(* IEC 61131-3 sources: axftcmlib/src/Actuator, 6 files *)

(* ---- ActuatorStates.st ---- *)
NAMESPACE Simatic.Ax.axftcmlib
    TYPE
        ActuatorState : (Retracted, Activating, Activated, Retracting) := Retracted;
    END_TYPE
END_NAMESPACE

(* ---- IActuator.st ---- *)
USING Simatic.Ax.Commands;
NAMESPACE Simatic.Ax.axftcmlib
    INTERFACE IActuator
        METHOD Start : itfCommand END_METHOD
    END_INTERFACE
END_NAMESPACE

(* ---- itfActuator.st ---- *)
USING Simatic.Ax.Commands;

NAMESPACE Simatic.Ax.axftcmlib

    INTERFACE itfActuator
        METHOD GoToWorkPosition : itfCommand
        END_METHOD
    END_INTERFACE

    INTERFACE itfTwoWayActuator EXTENDS itfActuator
        METHOD GoToHomePosition : itfCommand
        END_METHOD
    END_INTERFACE

END_NAMESPACE

(* ---- ActuatorTimeBased.st ---- *)
USING Simatic.Ax.Commands;
USING System.Timer;
USING Simatic.Ax.Io.Output;

NAMESPACE Simatic.Ax.axftcmlib
    CLASS ActuatorTimeBased
        EXTENDS ExecuteControlModuleAbstract
        IMPLEMENTS itfActuator
        VAR PUBLIC
            Q_ToWorkPosition : IBinOutput;
            OnDuration : TIME;
        END_VAR
        VAR
            _tonOnDuration : OnDelay;
            _state : ActuatorState;
        END_VAR

        METHOD PROTECTED OVERRIDE _initmethod
            ;
        END_METHOD

        METHOD PROTECTED OVERRIDE _executeCustom
            IF (Q_ToWorkPosition = NULL) THEN
                THIS.SetError(WORD#16#8101);
                RETURN;
            ELSE
                THIS.SetError(FALSE);
            END_IF;
            _tonOnDuration(signal := Q_ToWorkPosition.IsOn(), Duration := OnDuration);
            CASE _state OF
                // Switch all outputs off, when actuator is idle in home position
                ActuatorState#InHomePosition:
                    Q_ToWorkPosition.SetOff();

                // Received the command GoToWorkPosition switch on ToWorkPosition
                ActuatorState#MoveToWorkPosition:
                    Q_ToWorkPosition.SetOn();
                    _state := ActuatorState#InWorkPosition;
                // After Timeout switch off "ToWorkPosition"
                ActuatorState#InWorkPosition:
                    IF (_tonOnDuration.output) THEN
                        _state := ActuatorState#MoveToHomePosition;
                        Q_ToWorkPosition.SetOff();
                    END_IF;
                // Send done
                ActuatorState#MoveToHomePosition:
                    Q_ToWorkPosition.SetOff();
                    _state := ActuatorState#InHomePosition;
                    THIS.SetDone();
            END_CASE;
        END_METHOD

        METHOD PUBLIC GoToWorkPosition : itfCommand
            THIS.InitState();
            _state := ActuatorState#MoveToWorkPosition;
            GoToWorkPosition := THIS;
        END_METHOD

        METHOD PUBLIC GetState : ActuatorState
            GetState := _state;
        END_METHOD

    END_CLASS

END_NAMESPACE

(* ---- TimeBasedActuator.st ---- *)
USING Simatic.Ax.Commands;
USING System.Timer;
USING Simatic.Ax.Io.Output;

NAMESPACE Simatic.Ax.axftcmlib

    CLASS TimeBasedActuator
        EXTENDS ExecuteControlModuleAbstract
        IMPLEMENTS itfActuator
        VAR PUBLIC
            Q_ToWorkPosition : ItfBinOutput;
            OnDuration : TIME;
        END_VAR
        VAR
            _tonOnDuration : OnDelay;
            _state : ActuatorState;
        END_VAR

        METHOD PROTECTED OVERRIDE _initmethod
            ;
        END_METHOD

        METHOD PROTECTED OVERRIDE _executeCustom
            IF (Q_ToWorkPosition = NULL) THEN
                THIS.SetError(WORD#16#8101);
                RETURN;
            END_IF;
            _tonOnDuration(signal := Q_ToWorkPosition.IsOn(), Duration := OnDuration);
            CASE _state OF
// Switch all outputs off, when actuator is idle in home position
                ActuatorState#InHomePosition:
                    Q_ToWorkPosition.SetOff();
// Received the command GoToWorkPosition switch on ToWorkPosition
                ActuatorState#MoveToWorkPosition:
                    Q_ToWorkPosition.SetOn();
                    _state := ActuatorState#InWorkPosition;
// After Timeout switch off "ToWorkPosition"
                ActuatorState#InWorkPosition:
                    IF (_tonOnDuration.output) THEN
                        _state := ActuatorState#MoveToHomePosition;
                        Q_ToWorkPosition.SetOff();
                    END_IF;
// Send done
                ActuatorState#MoveToHomePosition:
                    Q_ToWorkPosition.SetOff();
                    _state := ActuatorState#InHomePosition;
                    THIS.SetDone();
            END_CASE;
        END_METHOD

        METHOD PUBLIC GoToWorkPosition : itfCommand
            THIS.InitState();
            _state := ActuatorState#MoveToWorkPosition;
            GoToWorkPosition := THIS;
        END_METHOD

        METHOD PUBLIC GetState : ActuatorState
            GetState := _state;
        END_METHOD
    END_CLASS

END_NAMESPACE

(* ---- TwoWayActuator.st ---- *)
USING Simatic.Ax.IO.Input;
USING Simatic.Ax.Commands;
USING System.Timer;
USING Simatic.Ax.Io.Output;

NAMESPACE Simatic.Ax.axftcmlib

    CLASS TwoWayActuator
        EXTENDS ActuatorTimeBased
        IMPLEMENTS itfTwoWayActuator
        VAR PUBLIC
            I_InHomePosition : IBinSignal;
            I_InWorkPosition : IBinSignal;
            Q_ToHomePosition : IBinOutput;
        END_VAR

        METHOD PROTECTED OVERRIDE _initmethod
            ;
        END_METHOD

        METHOD PROTECTED OVERRIDE _executeCustom
            IF (Q_ToWorkPosition = NULL) THEN
                THIS.SetError(WORD#16#8101);
                RETURN;
            ELSE
                THIS.SetError(FALSE);
            END_IF;
            CASE _state OF
                // Switch all outputs off, when actuator is idle in home position
                ActuatorState#InHomePosition:
                    Q_ToWorkPosition.SetOff();
                    Q_ToHomePosition.SetOff();
                // Received the command GoToWorkPosition switch on ToWorkPosition
                ActuatorState#MoveToWorkPosition:
                    Q_ToWorkPosition.SetOn();
                    IF (I_InWorkPosition.Q()) THEN
                        Q_ToWorkPosition.SetOff();
                        THIS.SetDone();
                        _state := ActuatorState#InWorkPosition;
                    END_IF;
                ActuatorState#InWorkPosition:
                    Q_ToWorkPosition.SetOff();
                    Q_ToHomePosition.SetOff();
                ActuatorState#MoveToHomePosition:
                    Q_ToHomePosition.SetOn();
                    IF (I_InHomePosition.Q()) THEN
                        Q_ToHomePosition.SetOff();
                        THIS.SetDone();
                        _state := ActuatorState#InHomePosition;
                        THIS.SetDone();
                    END_IF;
            END_CASE;
        END_METHOD

        METHOD PUBLIC GoToHomePosition : itfCommand
            THIS.InitState();
            _state := ActuatorState#MoveToHomePosition;
            GoToHomePosition := THIS;
        END_METHOD

    END_CLASS

END_NAMESPACE
